FUNCTION_BLOCK FB_BWK
VAR_INPUT
	Freigabe_auto			: BOOL;
	Freigabe_Deakt_auto		: BOOL;
	Betrieb_Anford_auto		: BOOL;
	Regelung_Modus_auto		: SINT;
	Regelung_Sollw_auto		: REAL;
	Quittierung				: BOOL;
	Parameter_init			: ST_BWK_Parameter;
END_VAR
VAR_OUTPUT
	{attribute 'OPC.UA.DA' := '1'}Steuerung				: ST_BWK_Steuerung;	
	{attribute 'OPC.UA.DA' := '1'}Stellwert				: ST_BWK_Stellwert;	
	{attribute 'OPC.UA.DA' := '1'}Zustand					: ST_BWK_Zustand;
	{attribute 'OPC.UA.DA' := '1'}Parameter				: ST_BWK_Parameter;	
END_VAR
VAR
	Zustandscheck			: FB_BWK_Zustandscheck;
	Logik					: FB_BWK_Logik;
	Ablaufsteuerung			: FB_BWK_Ablaufsteuerung;
	Sollwertscheck			: FB_BWK_Sollwertscheck;
	Regelung				: FB_BWK_Regelung;
	Stellwertscheck			: FB_BWK_Stellwertscheck;
	QuitTrig				: FB_SetResetFallTrigger;

(*	LeseDaten				: FB_BWK_Input;
	IN_Leistung				AT %I* : SINT;	(* 0..100 % *)
	IN_Temp_Ist				AT %I* : REAL;

	SchreibeDaten			: FB_BWK_Output;
	OUT_Betrieb				AT %Q* : BOOL;
	OUT_Modus				AT %Q* : SINT;
	OUT_Leistung			AT %Q* : SINT;
	OUT_Temperatur			AT %Q* : REAL;
*)

	Kommunikation			: LON_COM;

	OUT_Flow_T				: REAL := 0;
	OUT_Leistung			: SINT := 0;
	OUT_Temp_Soll			: REAL := 0;

	OUT_MODUS				: INT :=1; (*1=HVAC_HEAT   100=HVAC_FLOW_TEMP*)
	SchreibeDaten			: FB_BWK_SchreibeDaten;
	OUT_Stellung			AT %Q* : BOOL;
END_VAR

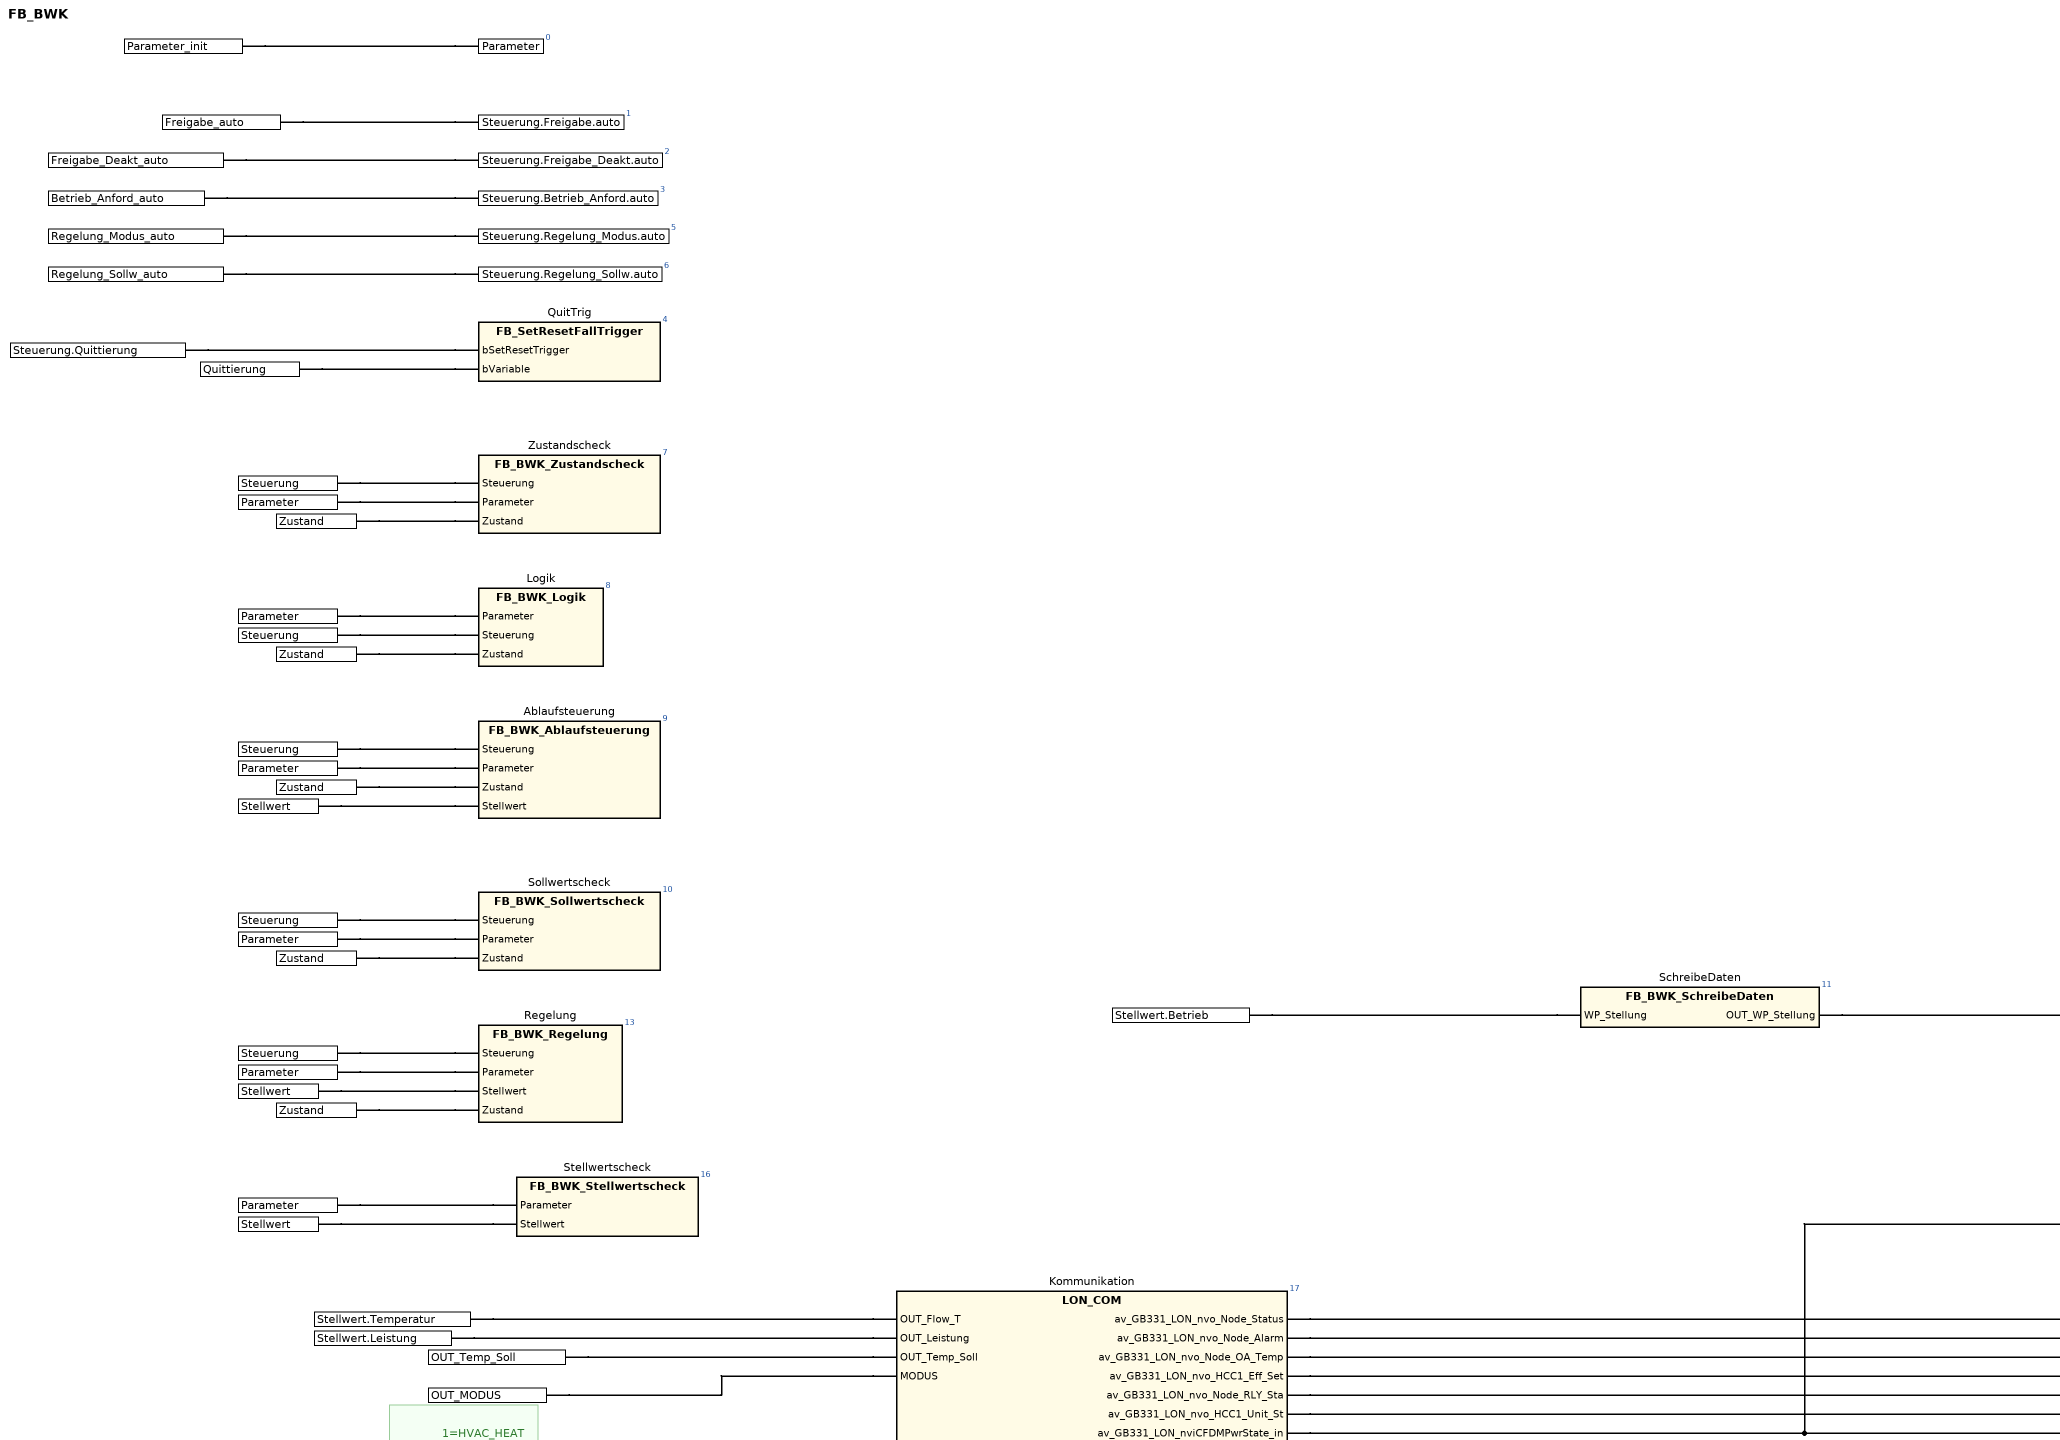
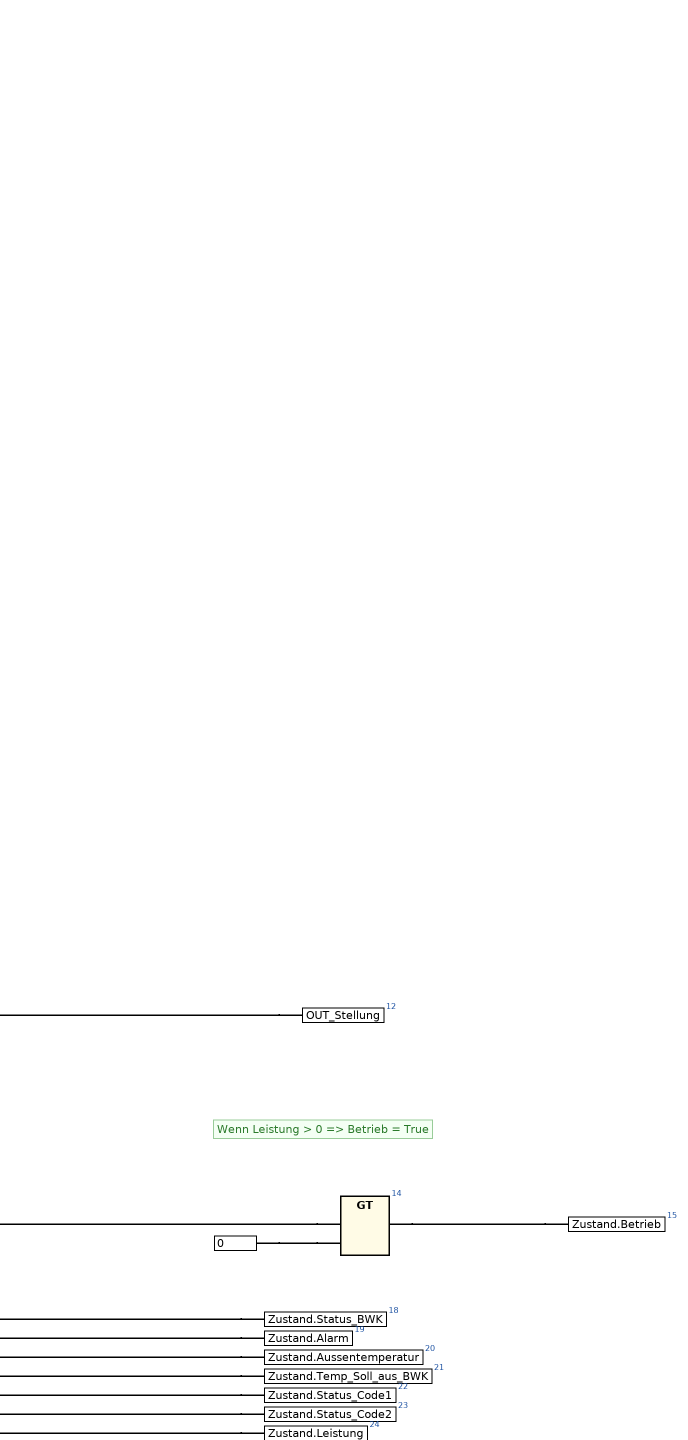
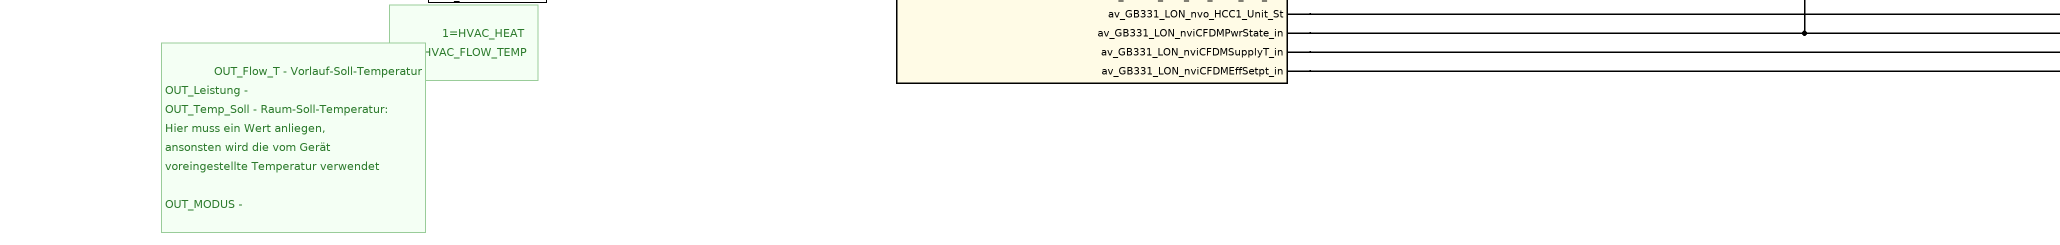
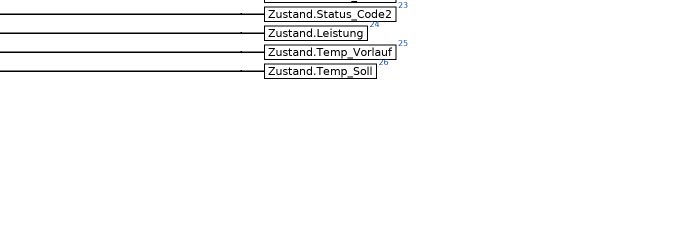
Parameter := Parameter_init;
Steuerung.Freigabe.auto := Freigabe_auto;
Steuerung.Freigabe_Deakt.auto := Freigabe_Deakt_auto;
Steuerung.Betrieb_Anford.auto := Betrieb_Anford_auto;
QuitTrig(bSetResetTrigger := Steuerung.Quittierung, bVariable := Quittierung); // FB_SetResetFallTrigger
Steuerung.Regelung_Modus.auto := Regelung_Modus_auto;
Steuerung.Regelung_Sollw.auto := Regelung_Sollw_auto;
Zustandscheck(Steuerung := Steuerung, Parameter := Parameter, Zustand := Zustand); // FB_BWK_Zustandscheck
Logik(Parameter := Parameter, Steuerung := Steuerung, Zustand := Zustand); // FB_BWK_Logik
Ablaufsteuerung(Steuerung := Steuerung, Parameter := Parameter, Zustand := Zustand, Stellwert := Stellwert); // FB_BWK_Ablaufsteuerung
Sollwertscheck(Steuerung := Steuerung, Parameter := Parameter, Zustand := Zustand); // FB_BWK_Sollwertscheck
SchreibeDaten(WP_Stellung := Stellwert.Betrieb); // FB_BWK_SchreibeDaten
OUT_Stellung := SchreibeDaten.OUT_WP_Stellung;
Regelung(Steuerung := Steuerung, Parameter := Parameter, Stellwert := Stellwert, Zustand := Zustand); // FB_BWK_Regelung
// Wenn Leistung > 0 => Betrieb = True
Zustand.Betrieb := Kommunikation.av_GB331_LON_nviCFDMPwrState_in > 0;
Stellwertscheck(Parameter := Parameter, Stellwert := Stellwert); // FB_BWK_Stellwertscheck
// 							1=HVAC_HEAT
// 100=HVAC_FLOW_TEMP
//
// 							OUT_Flow_T - Vorlauf-Soll-Temperatur
// OUT_Leistung -
// OUT_Temp_Soll - Raum-Soll-Temperatur:
// Hier muss ein Wert anliegen,
// ansonsten wird die vom Gerät
// voreingestellte Temperatur verwendet
//
// OUT_MODUS -
//
Kommunikation(
    OUT_Flow_T := Stellwert.Temperatur,
    OUT_Leistung := Stellwert.Leistung,
    OUT_Temp_Soll := OUT_Temp_Soll,
    MODUS := OUT_MODUS); // LON_COM
Zustand.Status_BWK := Kommunikation.av_GB331_LON_nvo_Node_Status;
Zustand.Alarm := Kommunikation.av_GB331_LON_nvo_Node_Alarm;
Zustand.Aussentemperatur := Kommunikation.av_GB331_LON_nvo_Node_OA_Temp;
Zustand.Temp_Soll_aus_BWK := Kommunikation.av_GB331_LON_nvo_HCC1_Eff_Set;
Zustand.Status_Code1 := Kommunikation.av_GB331_LON_nvo_Node_RLY_Sta;
Zustand.Status_Code2 := Kommunikation.av_GB331_LON_nvo_HCC1_Unit_St;
Zustand.Leistung := Kommunikation.av_GB331_LON_nviCFDMPwrState_in;
Zustand.Temp_Vorlauf := Kommunikation.av_GB331_LON_nviCFDMSupplyT_in;
Zustand.Temp_Soll := Kommunikation.av_GB331_LON_nviCFDMEffSetpt_in;

END_FUNCTION_BLOCK

(* stored: Version 1.1.0.1, ProductVersion 3.1.4024.9
   POU FB_BWK: Id {179f9f55-6990-4db2-ac35-92cac00747cd}, SpecialFunc None *)
